FUNCTION F_AnalogIntToVoltage : REAL
VAR_INPUT
	AnalogValue	: INT;
END_VAR
VAR
	Max_Int_Value_pos	: INT := 32767;
	Max_Int_Value_Neg	: INT := -32768;
	Voltagevalue 		: REAL := 10;
END_VAR



IF AnalogValue > 0 THEN
	F_AnalogIntToVoltage := Voltagevalue*(INT_TO_REAL(AnalogValue)/INT_TO_REAL(Max_Int_Value_pos));
ELSIF AnalogValue < 0 THEN
	F_AnalogIntToVoltage :=  Voltagevalue*(INT_TO_REAL(AnalogValue)/INT_TO_REAL(Max_Int_Value_Neg));
ELSE
	F_AnalogIntToVoltage := 0;
END_IF

END_FUNCTION

(* stored: Version 1.1.0.1, ProductVersion 3.1.4022.17
   POU F_AnalogIntToVoltage: Id {38787ad6-3d84-4540-ab0e-5b15702090f2}, SpecialFunc None *)
